FUNCTION TFLeastUsedCode : INT
VAR_INPUT
	EnableCode : ARRAY [1..MAXFORMINGCODE*MAXFORMING] OF INT;
	UsedCode : POINTER TO ARRAY [1..MAXFORMINGCODE] OF INT;
END_VAR
VAR
	Code : INT;
	i : INT;
	j : INT;
	Counter : INT;
	MinCounter : INT;
END_VAR

TFLeastUsedCode := 0;
Code := 0;
MinCounter := MAXFORMINGCODE + 1;

FOR i:=1 TO MAXFORMINGCODE*MAXFORMING DO
	IF EnableCode[i] > 0 THEN
		Counter := 0;
		FOR j:=1 TO MAXFORMINGCODE DO
			IF UsedCode^[j] = EnableCode[i] THEN
				Counter := Counter + 1;
			END_IF
		END_FOR
		IF Counter < MinCounter THEN
			MinCounter := Counter;
			Code := EnableCode[i];
		END_IF 
	END_IF
END_FOR

TFLeastUsedCode := Code;

END_FUNCTION

(* stored: Version 1.1.0.1, ProductVersion 3.1.4024.11
   POU TFLeastUsedCode: Id {c71060a1-1549-4b62-a9ac-5e8e8fdbd294}, SpecialFunc None *)
